Fanuc TP program (LS listing): _FLTLIM.LS

/PROG  _FLTLIM
/ATTR
OWNER		= MNEDITOR;
COMMENT		= "Limit Error";
PROG_SIZE	= 290;
CREATE		= DATE 21-03-19  TIME 11:14:44;
MODIFIED	= DATE 21-03-19  TIME 11:14:44;
FILE_NAME	= _FLTCOL;
VERSION		= 0;
LINE_COUNT	= 4;
MEMORY_SIZE	= 654;
PROTECT		= READ_WRITE;
TCD:  STACK_SIZE	= 0,
      TASK_PRIORITY	= 50,
      TIME_SLICE	= 0,
      BUSY_LAMP_OFF	= 0,
      ABORT_REQUEST	= 0,
      PAUSE_REQUEST	= 0;
DEFAULT_GROUP	= *,*,*,*,*;
CONTROL_CODE	= 00000000 00000000;
/APPL
/APPL
/MN
   1:  !***************************** ;
   2:  !Limit Error ;
   3:  !***************************** ;
   4:  CALL _FAULT(12) ;
/POS
/END
